{attribute 'linkalways'} 
{attribute 'no_explicit_call' := 'This FB is a CLASS and must be accessed using methods or properties'}
{attribute 'enable_dynamic_creation'}
FUNCTION_BLOCK _Array0to2OfUSINT EXTENDS ArrayDatatypeBase
VAR CONSTANT
	lBound : DINT := 0;
	uBound : DINT := 2;
END_VAR
VAR
	localData : ARRAY [lBound..uBound] OF USINT;
	activeData : REFERENCE TO ARRAY [lBound..uBound] OF USINT REF= localData;
	elements : ARRAY [lBound..uBound] OF _USINT(0);
	baseType : _USINT(0);
END_VAR

PROPERTY PUBLIC Address : PVOID
GET
Address := ADR(activeData);
END_GET
END_PROPERTY

PROPERTY PUBLIC BaseDatatype : I_Datatype
GET
BaseDatatype := baseType;
END_GET
END_PROPERTY

METHOD PUBLIC ClearReference
VAR_INPUT
END_VAR
activeData REF= localData;
SetElementReference();
END_METHOD

METHOD PUBLIC Clone : I_Datatype
VAR
    pClone : POINTER TO _Array0to2OfUSINT;
END_VAR
pClone := __NEW(_Array0to2OfUSINT());
pClone^.Value := Value;
Clone := pClone^;
END_METHOD

METHOD FB_init : BOOL
VAR_INPUT
	bInitRetains : BOOL; // if TRUE, the retain variables are initialized (warm start / cold start)
	bInCopyCode : BOOL;  // if TRUE, the instance afterwards gets moved into the copy code (online change)
END_VAR
SetElementReference();
END_METHOD

METHOD PUBLIC GetElementAsDatatypeByIndex : I_Datatype
VAR_INPUT
	Index : DINT;
END_VAR
GetElementAsDatatypeByIndex := elements[Index];
END_METHOD

METHOD PUBLIC GetElementByIndex : REFERENCE TO _USINT;
VAR_INPUT
	Index : DINT;
END_VAR
GetElementByIndex REF= elements[Index];
END_METHOD

PROPERTY PUBLIC LowerBound : DINT
GET
LowerBound := lBound;
END_GET
END_PROPERTY

METHOD PUBLIC MakeReferenceTo
VAR_INPUT
	ReferenceTarget : REFERENCE TO ARRAY [lBound..uBound] OF USINT;
END_VAR
activeData REF= ReferenceTarget;
SetElementReference();
END_METHOD

METHOD PROTECTED OnSerializeArrayValues
VAR_INPUT
	Serializer : I_Serializer;
END_VAR
VAR
	i : DINT;
END_VAR
FOR i := lBound TO uBound DO
	elements[i].SerializeWith(Serializer);
END_FOR
END_METHOD

METHOD PROTECTED SetElementReference
VAR_INPUT
END_VAR
VAR
	i : DINT;
END_VAR
FOR i := lBound TO uBound DO
	elements[i].MakeReferenceTo(activeData[i]);
END_FOR
END_METHOD

PROPERTY PUBLIC Size : UDINT
GET
Size := SIZEOF(activeData);
END_GET
END_PROPERTY

METHOD PROTECTED TryDeserializeArrayValues : BOOL
VAR_INPUT
	Deserializer : I_Deserializer;
	Feedback : I_DeserializerFeedback;
END_VAR
VAR
	enumerator : I_DeserializerArrayForwardEnumerator;
	i : DINT;
END_VAR
enumerator := Deserializer.GetArrayEnumerator();
i := lBound;

WHILE enumerator.MoveNext() AND i <= uBound DO
	
	IF NOT elements[i].TryDeserializeFrom(enumerator.Current, Feedback) THEN
		EXIT;
	END_IF
	i := i + 1;

END_WHILE
enumerator.Dispose();
END_METHOD

METHOD TryMakeReferenceTo : BOOL
VAR_INPUT
	Target : I_Datatype;
END_VAR
VAR
	targetAsArray : I_ArrayDatatype;
	pTargetData : POINTER TO ARRAY [lBound..uBound] OF USINT;
END_VAR
IF NOT Target.TryResolveAsArrayDatatype(targetAsArray) THEN
	RETURN;
END_IF

IF NOT (targetAsArray.Identifier = Identifier) THEN
	RETURN;
END_IF

pTargetData := Target.Address;
activeData REF= pTargetData^;
SetElementReference();
TryMakeReferenceTo := TRUE;
END_METHOD

PROPERTY PUBLIC UpperBound : DINT
GET
UpperBound := ubound;
END_GET
END_PROPERTY

PROPERTY PUBLIC Value : REFERENCE TO ARRAY [lBound..uBound] OF USINT;
GET
Value ref= activeData;
END_GET
END_PROPERTY

END_FUNCTION_BLOCK

(* stored: Version 1.1.0.1, ProductVersion 3.1.4024.13
   POU _Array0to2OfUSINT: Id {97ba6251-0797-08ad-20c4-a811d2a463cd}, SpecialFunc None
   Folder Core: Id {c8c2dcb0-0abc-09e6-0173-6104034d8f14}
   Folder Constructor: Id {0f0242f7-7a22-0f5d-3622-5f2729badf06}
   Folder Protected: Id {df16b176-f1ae-056f-3b88-479f5a635a61}
   Folder Customize: Id {0b04ff73-2076-0098-3463-8f276c6c7a5a}
   Property Address: Id {4a8c2627-9691-0984-07f6-e6a946cfc351}
   Get Get: Id {7cea8611-8b8c-0155-1f10-de1837effbe8}
   Property BaseDatatype: Id {a29f596c-908e-0435-38d2-f4b4d00d45cc}
   Get Get: Id {57591a66-4036-0aa3-340a-76e60e1a0696}
   Method ClearReference: Id {0e2bfd1a-ba93-0966-2cb9-8d6c137eca0c}
   Method Clone: Id {78cdaf05-3d2f-0d2e-1878-6b9e44e5057d}
   Method FB_init: Id {04d25559-214e-0e92-1b2c-2607f0566690}
   Method GetElementAsDatatypeByIndex: Id {4484af21-d08c-0e0f-19f4-bd8ecb9f5bbf}
   Method GetElementByIndex: Id {f2093af8-e723-0d00-3be5-99a84ae49236}
   Property LowerBound: Id {b9ebca3c-9ba8-0ccc-3615-afe9928f6061}
   Get Get: Id {6a2150a8-0988-0706-0a74-987479446aac}
   Method MakeReferenceTo: Id {3c225855-8ae7-0149-3ecf-9e8a1a5ab443}
   Method OnSerializeArrayValues: Id {44fac112-5a93-0230-08b6-f24e6bd03845}
   Method SetElementReference: Id {b8ddc947-8c17-0f20-1db8-5991f028b248}
   Property Size: Id {2fd77a84-a7f2-0e2d-2c9c-775b51528763}
   Get Get: Id {3a3210e9-bb46-063b-31e2-0aeea18d0771}
   Method TryDeserializeArrayValues: Id {2db53d5e-2ea9-0a47-1679-f7ca7ee854d0}
   Method TryMakeReferenceTo: Id {b3a722ae-c8ae-0410-26b5-ca5c2e4fd661}
   Property UpperBound: Id {f828136b-4570-061e-2cca-38e9f789c216}
   Get Get: Id {e6697fbb-84ea-0ee0-2a9b-930af03409c0}
   Property Value: Id {0b3cb14b-e52a-0865-0a82-426d566d3bd0}
   Get Get: Id {9695706b-6b33-0379-3cc2-86199b0683b0} *)
